// TIA Portal V15.1 export
// export: Created 2024-05-17T05:38:27.7173353Z, ExportSetting WithDefaults, DisplayName Totally Integrated Automation Portal, DisplayVersion V15.1 Update 5, DisplayName TIA Portal Openness, DisplayVersion V15.1 Update 5, DisplayName SINAMICS Startdrive Advanced, DisplayVersion V15.1, DisplayName G130, G150, S120, S150, SINAMICS MV, S210, DisplayVersion V15.1, DisplayName G110M, G120, G120C, G120D, G120P, DisplayVersion V15.1, DisplayName STEP 7 Professional, DisplayVersion V15.1 Update 5, DisplayName STEP 7 Safety, DisplayVersion V15.1, DisplayName WinCC Professional, DisplayVersion V15.1 Update 5, DisplayName SIMATIC Visualization Architect, DisplayVersion V15.1
FUNCTION "LETAFuseModule25_32_CPC20PN-Config" : Void   // FC1409, SCL
{ S7_Optimized_Access := 'TRUE' }
VERSION : 0.1
// stored: AutoNumber false, IsIECCheckEnabled false, SetENOAutomatically False, UDAEnableTagReadback false
   VAR_INPUT
      I_FuseMod25_Used : Bool;   // Fuse module is used
      I_FuseMod25_CH1_NominalCurrent : Int;   // Nominal current for the fuse
      I_FuseMod25_CH1_Name : String;   // Fuse name
      I_FuseMod25_CH1_Description : String;   // Description
      I_FuseMod25_CH2_NominalCurrent : Int;   // Nominal current for the fuse
      I_FuseMod25_CH2_Name : String;   // Fuse name
      I_FuseMod25_CH2_Description : String;   // Description
      I_FuseMod26_Used : Bool;   // Fuse module is used
      I_FuseMod26_CH1_NominalCurrent : Int;   // Nominal current for the fuse
      I_FuseMod26_CH1_Name : String;   // Fuse name
      I_FuseMod26_CH1_Description : String;   // Description
      I_FuseMod26_CH2_NominalCurrent : Int;   // Nominal current for the fuse
      I_FuseMod26_CH2_Name : String;   // Fuse name
      I_FuseMod26_CH2_Description : String;   // Description
      I_FuseMod27_Used : Bool;   // Fuse module is used
      I_FuseMod27_CH1_NominalCurrent : Int;   // Nominal current for the fuse
      I_FuseMod27_CH1_Name : String;   // Fuse name
      I_FuseMod27_CH1_Description : String;   // Description
      I_FuseMod27_CH2_NominalCurrent : Int;   // Nominal current for the fuse
      I_FuseMod27_CH2_Name : String;   // Fuse name
      I_FuseMod27_CH2_Description : String;   // Description
      I_FuseMod28_Used : Bool;   // Fuse module is used
      I_FuseMod28_CH1_NominalCurrent : Int;   // Nominal current for the fuse
      I_FuseMod28_CH1_Name : String;   // Fuse name
      I_FuseMod28_CH1_Description : String;   // Description
      I_FuseMod28_CH2_NominalCurrent : Int;   // Nominal current for the fuse
      I_FuseMod28_CH2_Name : String;   // Fuse name
      I_FuseMod28_CH2_Description : String;   // Description
      I_FuseMod29_Used : Bool;   // Fuse module is used
      I_FuseMod29_CH1_NominalCurrent : Int;   // Nominal current for the fuse
      I_FuseMod29_CH1_Name : String;   // Fuse name
      I_FuseMod29_CH1_Description : String;   // Description
      I_FuseMod29_CH2_NominalCurrent : Int;   // Nominal current for the fuse
      I_FuseMod29_CH2_Name : String;   // Fuse name
      I_FuseMod29_CH2_Description : String;   // Description
      I_FuseMod30_Used : Bool;   // Fuse module is used
      I_FuseMod30_CH1_NominalCurrent : Int;   // Nominal current for the fuse
      I_FuseMod30_CH1_Name : String;   // Fuse name
      I_FuseMod30_CH1_Description : String;   // Description
      I_FuseMod30_CH2_NominalCurrent : Int;   // Nominal current for the fuse
      I_FuseMod30_CH2_Name : String;   // Fuse name
      I_FuseMod30_CH2_Description : String;   // Description
      I_FuseMod31_Used : Bool;   // Fuse module is used
      I_FuseMod31_CH1_NominalCurrent : Int;   // Nominal current for the fuse
      I_FuseMod31_CH1_Name : String;   // Fuse name
      I_FuseMod31_CH1_Description : String;   // Description
      I_FuseMod31_CH2_NominalCurrent : Int;   // Nominal current for the fuse
      I_FuseMod31_CH2_Name : String;   // Fuse name
      I_FuseMod31_CH2_Description : String;   // Description
      I_FuseMod32_Used : Bool;   // Fuse module is used
      I_FuseMod32_CH1_NominalCurrent : Int;   // Nominal current for the fuse
      I_FuseMod32_CH1_Name : String;   // Fuse name
      I_FuseMod32_CH1_Description : String;   // Description
      I_FuseMod32_CH2_NominalCurrent : Int;   // Nominal current for the fuse
      I_FuseMod32_CH2_Name : String;   // Fuse name
      I_FuseMod32_CH2_Description : String;   // Description
   END_VAR
   VAR_IN_OUT
      IO_Config : "ETAFuseCPC20PNConfig";
   END_VAR
BEGIN
   #IO_Config.Fuse[49].Used := #I_FuseMod25_Used;
   #IO_Config.Fuse[49].NominalCurrent := #I_FuseMod25_CH1_NominalCurrent;
   #IO_Config.Fuse[49].Name := #I_FuseMod25_CH1_Name;
   #IO_Config.Fuse[49].Description := #I_FuseMod25_CH1_Description;

   #IO_Config.Fuse[50].Used := #I_FuseMod25_Used;
   #IO_Config.Fuse[50].NominalCurrent := #I_FuseMod25_CH2_NominalCurrent;
   #IO_Config.Fuse[50].Name := #I_FuseMod25_CH2_Name;
   #IO_Config.Fuse[50].Description := #I_FuseMod25_CH2_Description;

   #IO_Config.Fuse[51].Used := #I_FuseMod26_Used;
   #IO_Config.Fuse[51].NominalCurrent := #I_FuseMod26_CH1_NominalCurrent;
   #IO_Config.Fuse[51].Name := #I_FuseMod26_CH1_Name;
   #IO_Config.Fuse[51].Description := #I_FuseMod26_CH1_Description;

   #IO_Config.Fuse[52].Used := #I_FuseMod26_Used;
   #IO_Config.Fuse[52].NominalCurrent := #I_FuseMod26_CH2_NominalCurrent;
   #IO_Config.Fuse[52].Name := #I_FuseMod26_CH2_Name;
   #IO_Config.Fuse[52].Description := #I_FuseMod26_CH2_Description;

   #IO_Config.Fuse[53].Used := #I_FuseMod27_Used;
   #IO_Config.Fuse[53].NominalCurrent := #I_FuseMod27_CH1_NominalCurrent;
   #IO_Config.Fuse[53].Name := #I_FuseMod27_CH1_Name;
   #IO_Config.Fuse[53].Description := #I_FuseMod27_CH1_Description;

   #IO_Config.Fuse[54].Used := #I_FuseMod27_Used;
   #IO_Config.Fuse[54].NominalCurrent := #I_FuseMod27_CH2_NominalCurrent;
   #IO_Config.Fuse[54].Name := #I_FuseMod27_CH2_Name;
   #IO_Config.Fuse[54].Description := #I_FuseMod27_CH2_Description;

   #IO_Config.Fuse[55].Used := #I_FuseMod28_Used;
   #IO_Config.Fuse[55].NominalCurrent := #I_FuseMod28_CH1_NominalCurrent;
   #IO_Config.Fuse[55].Name := #I_FuseMod28_CH1_Name;
   #IO_Config.Fuse[55].Description := #I_FuseMod28_CH1_Description;

   #IO_Config.Fuse[56].Used := #I_FuseMod28_Used;
   #IO_Config.Fuse[56].NominalCurrent := #I_FuseMod28_CH2_NominalCurrent;
   #IO_Config.Fuse[56].Name := #I_FuseMod28_CH2_Name;
   #IO_Config.Fuse[56].Description := #I_FuseMod28_CH2_Description;

   #IO_Config.Fuse[57].Used := #I_FuseMod29_Used;
   #IO_Config.Fuse[57].NominalCurrent := #I_FuseMod29_CH1_NominalCurrent;
   #IO_Config.Fuse[57].Name := #I_FuseMod29_CH1_Name;
   #IO_Config.Fuse[57].Description := #I_FuseMod29_CH1_Description;

   #IO_Config.Fuse[58].Used := #I_FuseMod29_Used;
   #IO_Config.Fuse[58].NominalCurrent := #I_FuseMod29_CH2_NominalCurrent;
   #IO_Config.Fuse[58].Name := #I_FuseMod29_CH2_Name;
   #IO_Config.Fuse[58].Description := #I_FuseMod29_CH2_Description;

   #IO_Config.Fuse[59].Used := #I_FuseMod30_Used;
   #IO_Config.Fuse[59].NominalCurrent := #I_FuseMod30_CH1_NominalCurrent;
   #IO_Config.Fuse[59].Name := #I_FuseMod30_CH1_Name;
   #IO_Config.Fuse[59].Description := #I_FuseMod30_CH1_Description;

   #IO_Config.Fuse[60].Used := #I_FuseMod30_Used;
   #IO_Config.Fuse[60].NominalCurrent := #I_FuseMod30_CH2_NominalCurrent;
   #IO_Config.Fuse[60].Name := #I_FuseMod30_CH2_Name;
   #IO_Config.Fuse[60].Description := #I_FuseMod30_CH2_Description;

   #IO_Config.Fuse[61].Used := #I_FuseMod31_Used;
   #IO_Config.Fuse[61].NominalCurrent := #I_FuseMod31_CH1_NominalCurrent;
   #IO_Config.Fuse[61].Name := #I_FuseMod31_CH1_Name;
   #IO_Config.Fuse[61].Description := #I_FuseMod31_CH1_Description;

   #IO_Config.Fuse[62].Used := #I_FuseMod31_Used;
   #IO_Config.Fuse[62].NominalCurrent := #I_FuseMod31_CH2_NominalCurrent;
   #IO_Config.Fuse[62].Name := #I_FuseMod31_CH2_Name;
   #IO_Config.Fuse[62].Description := #I_FuseMod31_CH2_Description;

   #IO_Config.Fuse[63].Used := #I_FuseMod32_Used;
   #IO_Config.Fuse[63].NominalCurrent := #I_FuseMod32_CH1_NominalCurrent;
   #IO_Config.Fuse[63].Name := #I_FuseMod32_CH1_Name;
   #IO_Config.Fuse[63].Description := #I_FuseMod32_CH1_Description;

   #IO_Config.Fuse[64].Used := #I_FuseMod32_Used;
   #IO_Config.Fuse[64].NominalCurrent := #I_FuseMod32_CH2_NominalCurrent;
   #IO_Config.Fuse[64].Name := #I_FuseMod32_CH2_Name;
   #IO_Config.Fuse[64].Description := #I_FuseMod32_CH2_Description;
END_FUNCTION
